// TIA Portal V20 export
// export: Created 2025-12-01T14:57:23.1812812Z, ExportSetting None, DisplayName Totally Integrated Automation Portal, DisplayVersion V20 Update 3, DisplayName TIA Portal Openness, DisplayVersion V20 Update 3, DisplayName TIA Portal Version Control Interface, DisplayVersion V20 Update 3, DisplayName STEP 7 Professional, DisplayVersion V20 Update 3, DisplayName STEP 7 Safety, DisplayVersion V20 Update 2, DisplayName WinCC Basic/Comfort/Advanced, DisplayVersion V20 Update 3, DisplayName WinCC Professional, DisplayVersion V20 Update 3, DisplayName WinCC Unified, DisplayVersion V20 Update 3
DATA_BLOCK "DB913_Router_DestinoDesvio"   // DB913
{ S7_Optimized_Access := 'FALSE' }
AUTHOR : ROUTER
NAME : 20130623
VERSION : 3.0
// stored: AutoNumber false
   VAR RETAIN
      DestinoDesvios { S7_SetPoint := 'True'} : Array[0.."ROUT_Max_Destinos"] of "ROUT_Destino_Desvios";   // Relacion de los Desvios Definidos por Destino
   END_VAR
BEGIN
END_DATA_BLOCK
